INTERFACE Cyclic EXTENDS Queryable

METHOD Cyclic
END_METHOD

END_INTERFACE

(* stored: Version 1.1.0.1
   Itf Cyclic: Id {6715db9d-9390-03be-1292-a6e9996f2bd7}
   Method Cyclic: Id {ab22785f-988f-0a49-15aa-f59bebb11b3e} *)
